PROGRAM PLC_PRG
VAR
	
	//Visualisation buttons	
	mxButtonReset	: BOOL;	
	mxButtonStart: BOOL;

	//Internal use
	mxStart: BOOL;
	mxDone: BOOL;
	mxComBusy: BOOL;
	CommData: CommunicationData;
	

	//Motion Function Blocks
	fbCommunicator: Communicator;

	fbABBGoToHome_1: ABBGoToHome;
	fbABBGoToStorage_1: ABBGoToStorage;
	fbABBPickLeaveStorage_1: ABBPickLeaveStorage;
	fbABBGoToHome_2: ABBGoToHome;
	fbABBPickLeaveConveyor1_1: ABBPickLeaveConveyor1;
	fbTON_1: TON;
	ABBProcessAssembly_0: ABBProcessAssembly;

END_VAR

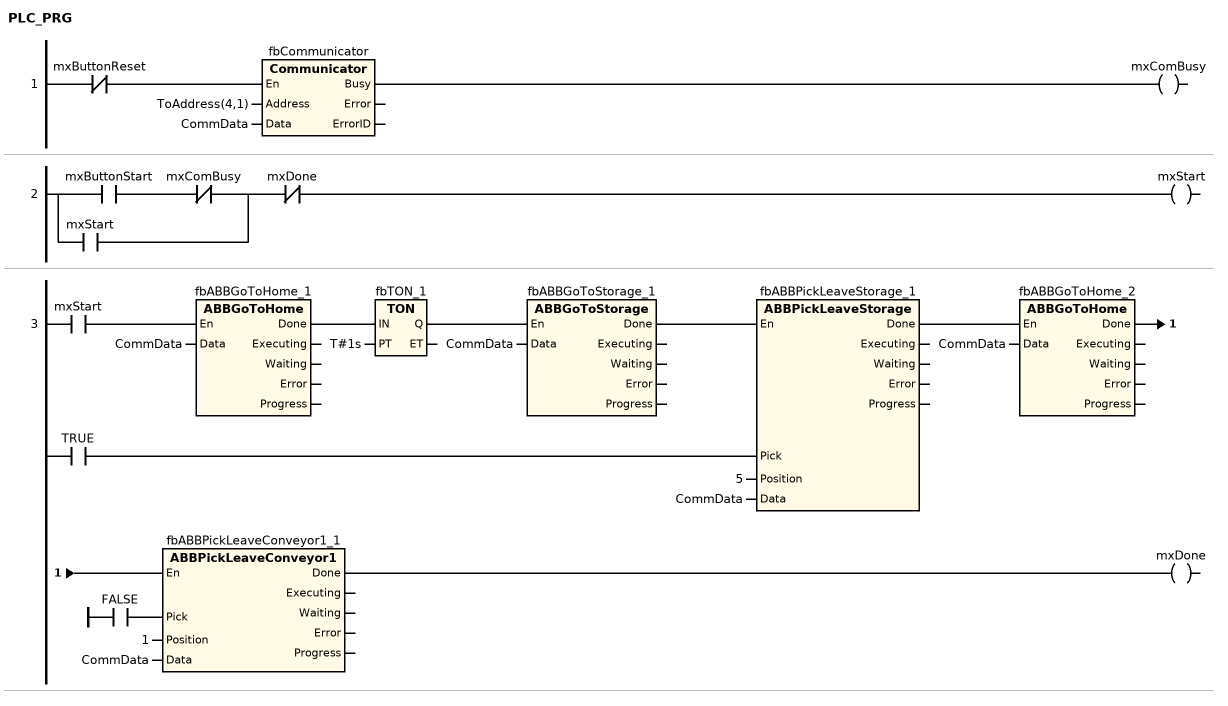
// NETWORK 1
fbCommunicator(En := NOT mxButtonReset, Address := ToAddress(4,1), Data := CommData); // Communicator
mxComBusy := fbCommunicator.Busy;

// NETWORK 2
mxStart := (mxButtonStart AND NOT mxComBusy OR mxStart) AND NOT mxDone;

// NETWORK 3
fbABBGoToHome_1(En := mxStart, Data := CommData); // ABBGoToHome
fbTON_1(IN := fbABBGoToHome_1.Done, PT := T#1s); // TON
fbABBGoToStorage_1(En := fbTON_1.Q, Data := CommData); // ABBGoToStorage
fbABBPickLeaveStorage_1(En := fbABBGoToStorage_1.Done, Pick := TRUE, Position := 5, Data := CommData); // ABBPickLeaveStorage
fbABBGoToHome_2(En := fbABBPickLeaveStorage_1.Done, Data := CommData); // ABBGoToHome
fbABBPickLeaveConveyor1_1(En := fbABBGoToHome_2.Done, Pick := FALSE, Position := 1, Data := CommData); // ABBPickLeaveConveyor1
mxDone := fbABBPickLeaveConveyor1_1.Done;

END_PROGRAM

(* stored: Version 1.1.0.1, ProductVersion 3.1.4022.12
   POU PLC_PRG: Id {6881d99a-5d83-480a-bf13-c68756a3bf82}, SpecialFunc None *)
